Staubli VAL3: print.pgx

public program print()
begin
  putln("robot_id: "+toString("",body.robotId))
  putln("sequence: "+toString("",body.sequence))
  putln("valid_fields: "+toString("",body.validFields))
  if bAnd(body.validFields,1)==1
    putln("time: "+toString(".3",body.time))
  endIf
  if bAnd(body.validFields,2)==2
    put("positions: ")
    call printArray("1.2",body.positions)
  endIf
  if bAnd(body.validFields,4)==4
    put("velocities: ")
    call printArray("1.2",body.velocities)
  endIf
  if bAnd(body.validFields,8)==8
    put("accelerations: ")
    call printArray("1.2",body.accelerations)
  endIf
end
